SUBAPPLICATION logiBUS_QXA_OPC (* logiBUS DQ Kanal: OPC-UA Read/Write (generisch, ein Kanal, ohne VT-Button/Hintergrundfarbe - fuer Module ohne ISOBUS/VT-Anbindung) *)
  (* Standard: 61499-2 *)
  (* Version 1.0, 2026-08-27, franz, Meisterschulen am Ostbahnhof *)
  PACKAGE MyLib::sys;
  IMPORT logiBUS::io::DQ::logiBUS_DO;
  IMPORT logiBUS::io::DQ::logiBUS_DO_S;
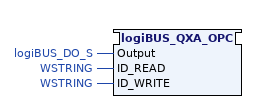
  VAR_INPUT
    Output : logiBUS::io::DQ::logiBUS_DO_S := logiBUS_DO::Invalid; (* Identify the Output Output_Q1..Q12 *)
    ID_READ : WSTRING; (* OPC-UA Subscribe-Key (schreibbar) *)
    ID_WRITE : WSTRING; (* OPC-UA Publish-Key (lesbar) *)
  END_VAR
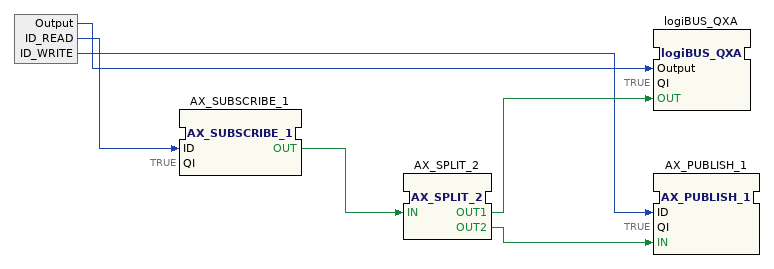
  FBS
    logiBUS_QXA : logiBUS::io::DQ::logiBUS_QXA(QI := TRUE);
    AX_SUBSCRIBE_1 : adapter::net::AX_SUBSCRIBE_1(QI := TRUE);
    AX_SPLIT_2 : adapter::events::unidirectional::AX_SPLIT_2;
    AX_PUBLISH_1 : adapter::net::AX_PUBLISH_1(QI := TRUE);
  END_FBS
  DATA_CONNECTIONS
    Output TO logiBUS_QXA.Output;
    ID_READ TO AX_SUBSCRIBE_1.ID;
    ID_WRITE TO AX_PUBLISH_1.ID;
  END_CONNECTIONS
  ADAPTER_CONNECTIONS
    AX_SUBSCRIBE_1.OUT TO AX_SPLIT_2.IN;
    AX_SPLIT_2.OUT1 TO logiBUS_QXA.OUT;
    AX_SPLIT_2.OUT2 TO AX_PUBLISH_1.IN;
  END_CONNECTIONS
END_SUBAPPLICATION
